{attribute 'linkalways'} 
{attribute 'no_explicit_call' := 'This FB is a CLASS and must be accessed using methods or properties'}
{attribute 'enable_dynamic_creation'}
FUNCTION_BLOCK FINAL EQ_ULINT EXTENDS Node
VAR
	in1 : _ULINT(0);
	in2 : _ULINT(0);
	out : _BOOL(FALSE);
END_VAR

METHOD PUBLIC Clone : I_Node
VAR
	pNode : POINTER TO EQ_ULINT;
END_VAR
pNode := __NEW(EQ_ULINT);
Clone := pNode^;
END_METHOD

METHOD FB_init : BOOL
VAR_INPUT
	bInitRetains : BOOL; // if TRUE, the retain variables are initialized (warm start / cold start)
	bInCopyCode : BOOL;  // if TRUE, the instance afterwards gets moved into the copy code (online change)
END_VAR
AddInput('in1',THIS^.in1);
AddInput('in2',THIS^.in2);
AddOutput('out', THIS^.out);
END_METHOD

METHOD PROTECTED OnExecute
VAR
END_VAR
out.Value := in1.Value = in2.Value;
END_METHOD

END_FUNCTION_BLOCK

(* stored: Version 1.1.0.1, ProductVersion 3.1.4024.15
   POU EQ_ULINT: Id {d8b6c169-7d02-4c3e-b06d-5dbaeb6a4784}, SpecialFunc None
   Folder Constructor: Id {562eddf7-5766-4896-be69-ab5c86df92d5}
   Method Clone: Id {355449b0-fd63-48b3-895f-c6e3764e70e8}
   Method FB_init: Id {d45e6770-8ab0-49d0-ba6a-7b83fc9cd759}
   Method OnExecute: Id {03253b30-ba9f-4256-9dc8-f745ca53a23e} *)
